// TIA Portal V21 export
TYPE "Std_stMotore"
   STRUCT
      In : Struct
         Setup : Bool;
         CmdPosRich : Bool;
         CmdNegRich : Bool;
         Positioning : Bool;
         PosRelativo : Bool;
         CambioVelDaPunto : Bool;
         ConsMovimentoPos : Bool;
         ConsMovimentoNeg : Bool;
         Premagnetizza : Bool;
         PremagnetizzaPos : Bool;
         PremagnetizzaNeg : Bool;
         ForzaEndLessPos : Bool;
         ForzaEndLessNeg : Bool;
         ForzaEndLessBreve : Bool;
         AttivaLimVarPos : Bool;
         AttivaLimVarNeg : Bool;
         MotoreRun : Bool;
         FrenoSganciato : Bool;
         AnticadutaON : Bool;
         AnticadutaOFF : Bool;
         CinghiaRotta : Bool;
         CoppiaSuperata : Bool;   // Ingresso digitale di coppia superata
         SezAperto : Bool;   // Ingresso digitale per sezionatore motore
         TerMotoreOff : Bool;   // Scatto termico motore
         TerVentolaOff : Bool;   // Scatto termico della servoventola
         DriverFault : Bool;   // Ingresso digitale per fault inverter
         DriverWarning : Bool;
         NoComunInv : Bool;
         NoComunEnc : Bool;
         SensAzz : Bool;
         SpinaSicNoInPos : Bool;
         IngInv01 : Bool;
         IngInv02 : Bool;
         IngInv03 : Bool;
         IngInv04 : Bool;
         IngInv05 : Bool;
         IngInv06 : Bool;
         IngInv07 : Bool;
         IngInv08 : Bool;
         PercentualeRichiesta : Int := 100;
         TrgPos : DInt;
         TrgPosRel : DInt;
         CmdVelocitaRich : DInt;
         Acc : DInt;
         Dec : DInt;
         PosCambioVel : DInt;
         VelCambioVel : DInt;
         LimiteVarPos : DInt;
         LimiteVarNeg : DInt;
         ValoSetupEnc : DInt;
      END_STRUCT;
      HW : Struct
         TipoCollInverter : Int;
         HWIO_Inverter : HW_IO;
         HWIO_Parametri : HW_IO;
         HWIO_Inverter_Out : HW_IO;
         HWIO_Parametri_Out : HW_IO;
         TipoEncoder : Int;
         HWIO_Encoder : HW_IO;
         HWIO_PrmEncoder : HW_IO;
      END_STRUCT;
      Prm : Struct
         Quote : Array[0.."K_NumCamma"] of Real;
         UnitàMisura : "Std_UnitàDiMisura";
         Mech : Struct
            Direction : Bool;
            EndLess : Bool;
            GearIn : UInt;
            GearOut : UInt;
            FeedConstant : UDInt;
            RPMMaxRef : UInt;
            JLoad : DInt;
            Z176 : DInt;
         END_STRUCT;
         Enc : Struct
            Direction : Bool;
            EncoderLess : Bool;
            Z180_2 : Bool;
            Z180_3 : Bool;
            Z180_4 : Bool;
            Z180_5 : Bool;
            Z180_6 : Bool;
            Z180_7 : Bool;
            ModoCalcoloK : Bool;
            SetupDoppio : Bool;
            Z181_2 : Bool;
            Z181_3 : Bool;
            Z181_4 : Bool;
            Z181_5 : Bool;
            Z181_6 : Bool;
            Z181_7 : Bool;
            Mounting : USInt;
            SetupMode : USInt;
            ModuloPosEnc : DInt := DINT#1_000_000_000;
            ModuloNegEnc : DInt;
            KSetup : DInt;
            FeedConstant : UDInt;
            ImpRev : Real;
         END_STRUCT;
         C : Struct
            ContPrema : Int;
            OldPosEncoder : DInt;
            TrgPos : Real;
            SpazioGiroEncoder : Real;
            EncPos : Real;
            VelMax : DInt;
         END_STRUCT;
         "M" : Struct
            RichManPos : Bool;
            RichManNeg : Bool;
            AsseNuovaPosManRich : Bool;
         END_STRUCT;
         AbiltManutenzionePrev : Bool;
         K_Analogica : Int;
         EscludiFunzPos : Bool;
         CalcTempoRimanente : Bool;
         CambioDirNoFreno : Bool;
         PremaNoFreno : Bool;
         FrenoPresente : Bool;
         FBKFrenoPresente : Bool;
         AnticadutaPresente : Bool;
         ByPassAnticaduta : Bool;
         DisabCicloAutoAllarme : Bool;
         DisabCicloManuAllarme : Bool;
         TReazioneSistema : Int := 120;
         TPrema : Int := 250;
         TBassaVel : Int := 100;
         TAggancioFreno : Int := 100;
         TSgancioFreno : Int := 100;
         TOutPrema : Int := 1000;
         TMinVCost : Int;
         TCambioDir : Int;
         ValMaxRef : Int;
         LimitePos : DInt;
         LimiteNeg : DInt;
         PosManutenzione : DInt;
         VelPrema : DInt;
         VelBassa : DInt;
         VelSgancioFrenoPos : DInt;
         VelSgancioFrenoNeg : DInt;
         SpazioArrestoPos : DInt;
         SpazioArrestoNeg : DInt;
         Precisione : DInt;
         Inerzia : DInt;
         FollowingLimit : DInt;
         MaxCopia : DInt;
         DecFinale : DInt;
         DecEmergenza : DInt;
         Jerk : DInt;
         VelMan : DInt;
         VelJog : DInt;
      END_STRUCT;
      Dati : Struct
         BloccoRichiamato : Bool;
         InclusoInUnaSequenza : Bool;
         SetupPN : Struct
            Input : Struct
               REQ : Bool;
               ID : Bool;
               INDEX : Bool;
               LEN : Bool;
            END_STRUCT;
            Output : Struct
               DONE : Bool;
               BUSY : Bool;
               ERROR : Bool;
               STATUS : DWord;
            END_STRUCT;
         END_STRUCT;
         MP : Struct
            SpazioPercorso : DInt;
            TempoMovimento : DInt;
            ImpMarcia : Bool;
            ImpFreno : Bool;
            MetriPercorsi : DInt;
            MinutiLavorati : DInt;
            NAvviamenti : DInt;
            NSgancioFreno : DInt;
         END_STRUCT;
         MotorStop : Bool;
         ActVelPos : Bool;   // Velocità Positiva in Corso
         ActVelNeg : Bool;   // Velocità Negativa in Corso
         MotoreFermo : Bool;   // Motore fermo
         RitAggancioFreno : Bool;   // Memoria tempo aggancio freno trascorso
         CambioDirezioneAlVolo : Bool;   // Eseguito cambio direzione al volo
         SetupSensoreTrovato : Bool;   // Sensore di Setup Trovato
         SetupFermoMeccTrovato : Bool;   // Arresto meccanico durante procedura di Set Up Trovato
         TOffInverterStatus : Bool;   // Ritardo OFF segnale stato inverter
         TOffMotoreMarcia : Bool;   // Ritardo OFF Motore in Marcia
         AppoImpMotoreFermo : Bool;   // Appoggio Impulso motore fermo
         AppoImpEsecSetUP : Bool;   // Appoggio Impulso richiesta SetUP Sensore o Fermo Meccanico
         AppoImpOnSegnSonora : Bool;   // Appoggio Impulso ON Segnalazione Sonora
         AppoImpFunzPositioning : Bool;   // Appoggio Impulso Richiesta funzionamento in posizione
         AppoImpMovRelativo : Bool;   // Appoggio Impulso per richiesta movimento relativo
         AppoImpCaVelPunto : Bool;   // Impulso di cambio velocità da punto
         StatoFreno : Bool;   // Stato Freno
         PrmSend : Bool;
         ContMotoreInPrec : Int;   // Conteggio tempo di motore all'interno della precisione [ms]
         ContTimeOutInverter : Int;   // Contatore Time Out Inverter [ms]
         ContTimeOutFreno1 : Int;   // Contatore Time Out Freno 1 (Rilascio) [ms]
         ContTimeOutFreno2 : Int;   // Contatore Time Out Freno 2 (Sganciato inaspettatamente) [ms]
         ContSgancioFreno : Int;   // Contatore ritardo Sgancio [ms]
         ContAggancioFreno : Int;   // Contatore ritardo Aggancio [ms]
         ContTimeOutPrema : Int;   // Contatore Time Out premagnetizzazione [ms]
         ContTOffInverterStatus : Int;   // Contatore Ritardo OFF Segnale Inverter Status [ms]
         ContTOffMotoreMarcia : Int;   // Contatore Ritardo OFF Motore in Marcia [ms]
         ContCheckFollowError : Int;   // Contatore per il controllo progressivo del Following Error [ms]
         ContSetUPEncoder : Int;   // Contatore per l'esecuzione del SetUP Encoder
         Memo_PercentualeRich : Int;   // Memorizzo la percentuale di velocità richiesta
         ContTimeOutAzzeramento : Int;   // Contatore Time Out Ricerca Sensori Azzeramento [ms]
         ContTOutAnticaduta : Int;   // Contatore Time-Out Anticaduta
         RetVal_Read_Inv : Int;   // Ret Val funzione Lettura Profibus dall'Inverter
         RetVal_SCR_Inv : Int;   // Ret Val funzione Scrittura Profibus all'Inverter
         ContCambioDirPos : Int;   // Contatore per cambio direzione Positiva
         ContCambioDirNeg : Int;   // Contatore per cambio direzione Negativa
         ContOffSezAperto : Int;   // Contatore per controllo sezionatore aperto SEW
         ContSegnSetup : Int;   // Contatore per segnalazione Setup Eseguita
         ContTORichSetup : Int;   // Contatore Time-Out richiesta Setup
         ContAbilAccDopoCambioDir : Int;   // Contatore Abilitazione Accelerazione dopo Cambio Direzione
         ContFermoMeccTrovato : Int;   // Contatore Fermo Meccanico Trovato
         IdPrm : UInt;   // Contatore Scrittura Parametri
         TempoEsecuzioneProfilo : DInt;   // Tempo esecuzione Profilo [ms]
         ContTimeOutMovimento : DInt;   // Contatore Time Out Movimento Motore [ms]
         ChFol_SpazioEncoder : DInt;   // Check Following: Spazio percorso dall'encoder nel tempo di controllo [Unità]
         ChFol_SpazioTarget : DInt;   // Check Following: Spazio percorso dal target nel tempo di controllo [Unità]
         TRG_OLD_POS_Select : DInt;   // OLD Posizione di target filtrata
         PosizioneAlloStop : DInt;   // Memorizzazione della posizione al momento dell'arresto [Unità]
         PosizioneCheckDirezione : DInt;   // Memorizzazione della posizione per il controllo della direzione [Unità]
         VeloRichPerc : DInt;   // Velocità richiesta dopo calcolo percentuale [Unità/s]
         AccRichPerc : DInt;   // Accelerazione richiesta dopo calcolo percentuale [Unità/s/s]
         DecRichPerc : DInt;   // Decelerazione richiesta dopo calcolo percentuale [Unità/s/s]
         VeloDopoCambioRich : DInt;   // Velocità dopo cambio richiesta [Unità/s]
         TrgPosDint : DInt;   // Posizione di target (Valore Intero) [Unità]
         OldTrgPosDint : DInt;   // Ultima Posizione di target (Valore Intero) [Unità]
         OldEncoder : DInt;   // Ultima Posizione letta dell'encoder [Unità]
         Memo_Req_Vel : DInt;   // Memorizzo la velocità richiesta [Unità/s]
         Memo_Req_Acc : DInt;   // Memorizzo l'accelerazione richiesta [Unità/s/s]
         Memo_Req_Dec : DInt;   // Memorizzo la decelerazione richiesta [Unità/s/s]
         Memo_Req_Dec_Emergenza : DInt;   // Memorizzo la decelerazione d'emergenza richiesta [Unità/s/s]
         PosImpulsoSetup : DInt;   // Posizione dell'impulso del sensore di Setup o della posizione di Fermo Meccanico [Unità]
         DecReqInLavo : DInt;   // Decelerazione richiesta in lavorazione
         DecReqFinaleInLavo : DInt;   // Decelerazione finale richiesta in lavorazione
         DecReqEmergInLavo : DInt;   // Decelerazione finale richiesta in lavorazione
         MovRelRichiesto : DInt;   // Movimento relativo richiesto [Unità]
         MemoCheckInversione : DInt;   // Memoria Controllo Inversione
         MaxPosRicercaFermoMeccanico : DInt;   // Massima Posizione durante la ricerca del fermo meccanico
         ReqVelConv : Real;   // Velocità richiesta convertito in REAL [Unità]
         VeloMinConv : Real;   // Velocità minima convertita
         Encoder : Struct
            PrmEncSend : Bool;   // Parametro Encoder Inviati
            OLD_Senso_Rotazione : Bool;   // Appoggio ultimo senso di rotazione Impostato
            RichSetupEnc { ExternalAccessible := 'False'; ExternalVisible := 'False'; ExternalWritable := 'False'} : Bool;   // Richiesta Setup Encoder
            RetValRdEnc : Int;   // RetVal funzione di lettura encoder
            RetValScrEnc : Int;   // RetVal funzione di scrittura encoder
            RicircoloEncoder : DInt := 0;   // Valore di ricircolo Encoder
            MezzoRicircoloEncoder : DInt := 0;   // Valore di mezzo ricircolo Encoder
            o_OldPosEncoder : DInt;   // Ultima posizione Encoder registrata [Impulsi]
            OLD_Spazio_Giro_Encoder : Real;   // Appoggio l'ultimo spazio per giro encoder Impostato
            ValoKSetupSuSens : DInt;   // Valore K Per Setup su Sensore
         END_STRUCT;
         AlmInv_ResetInverter : Bool;   // Allarme Inverter: Reset Inverter
         Alm_ContAzzCont : DInt;   // Autoreset Allarmi: Contatore Azzeramento Contatore Allarmi
         AlmBloccato_Cont : DInt := 0;   // Allarmi Bloccato: Conteggio
         AlmInv_ToutReset : Int;   // Allarme Inverter: Time Out Reset
         AlmInv_Cont : DInt := 0;   // Allarme Inverter: Conteggio
         AlmInv_ContStorico : DInt := 0;   // Allarme Inverter: Conteggio Storico
         AlmInv_RitRestart : Int;   // Allarme Inverter: Ritardo Ripartenza
         AlmInv_StoricoCodici : Array[0..9] of DInt;   // Allarme Inverter: Storico Codici
      END_STRUCT;
      HMI : Struct
         Visibilita : Struct
            Servoventola : Bool;
         END_STRUCT;
         Param : Struct
            Read : Bool;
            Write : Bool;
            Save : Bool;
            FactoryInit : Bool;
            Init_Motor : Bool;
            ReadAll : Bool;
            Number : Int;
            SubNumber : Int;
            Value : DInt;
         END_STRUCT;
         Setup : Bool;
         PulsanteSetupPremuto : Bool;
         ManMov : Bool;
         UpdParam : Bool;
         UM : USInt;
         FBGestione : Int;
         IndexAreaAuto : UInt;
         Stato : USInt;
         ComandoRichiesto : USInt;
         STW1 : Word;
         STW2 : Word;
         STW3 : Word;
         CTW1 : Word;
         CTW2 : Word;
         CTW3 : Word;
         ValoreSetupEncoder : DInt;
         ValoreSetupRichiesto : DInt;
         ValoreSetupSensore : DInt;
         CodiceWarning : DInt;
         CodiceAllarme : DInt;
         ModoInizializza : USInt;
         ALM : Array[0..1] of Word;
      END_STRUCT;
      Allarmi : Struct
         "A" : Array[0.."K_NumAllarmiPerMotori"] of "Std_PrmAllarmeStd";
         WordHmi_1 { S7_SetPoint := 'True'} : Word;
         WordHmi_2 : Word;
         ComunInverter : Bool;
         ComunEncoder : Bool;
         TOutMarcia : Bool;
         ConteggioEnc : Bool;
         FolError : Bool;
         Bloccato : Bool;
         TroppoVeloce : Bool;
         Direzione : Bool;
         EncMismatch : Bool;
         TOUTMovimento : Bool;
         InverterFault : Bool;
         TermicoVentola : Bool;
         RotturaCinghia : Bool;
         TimeOutAnticaduta : Bool;
         Freno : Bool;
         Freno2 : Bool;
         TOUT_Azzeramento : Bool;
         MotoreNonParam : Bool;
         EncoderNonSetup : Bool;
         SetupEncoderEseg : Bool;
         InverterWarning : Bool;
         Parametri : Bool;
         SezAperto : Bool;
         SpinaSicNoInPos : Bool;
         TrgPosMinNeg : Bool;
         TrgPosMaxPos : Bool;
         TrgPosMinNegVar : Bool;
         TrgPosMaxPosVar : Bool;
         AccRichZero : Bool;
         AccRichMaxMaxDec : Bool;
         DecRichZero : Bool;
         DecRichMaxMaxDec : Bool;
         DecFinaleRichZero : Bool;
         DecFinaleRichMaxMaxDec : Bool;
         DecEmergenzaRichZero : Bool;
         TrgVelMinFreno : Bool;
         TrgVelMaxMax : Bool;
         TrgVelCamMinFreno : Bool;
         TrgVelCamMaxMax : Bool;
      END_STRUCT;
      Out : Struct
         Pronto : Bool;
         PremaOK : Bool;
         TOUTPrema : Bool;
         InMarcia : Bool;
         ActDirPos : Bool;
         ActDirNeg : Bool;
         FaseAcc : Bool;
         FaseDec : Bool;
         PosOK : Bool;
         RichMovPos : Bool;
         RichMovNeg : Bool;
         MinLimNeg : Bool;
         MaxLimPos : Bool;
         ActInInerzia : Bool;
         MinTrg : Bool;
         MaxTrg : Bool;
         CmdPosServoventola : Bool;
         CmdPosMotore : Bool;
         CmdNegMotore : Bool;
         CmdAnticaduta : Bool;
         CmdFreno : Bool;
         RitSgancioFreno : Bool;
         Allarme : Bool;
         DisContattori : Bool;
         Lampada : Bool;
         Sirena : Bool;
         EncoderHomed : Bool;
         SetUpSensEseg : Bool;
         UpdParam : Bool;
         CmdUsc01Inv : Bool;
         CmdUsc02Inv : Bool;
         CmdUsc03Inv : Bool;
         CmdUsc04Inv : Bool;
         Paw : Word;
         ActPos : DInt;
         SpazioStop : DInt;
         ActPosPiuStop : DInt;
         ActPosPiuInerzia : DInt;
         ActPosMenoInerzia : DInt;
         SpazioCicloEnc : DInt;
         DistTRG : DInt;
         TrgPosFiltrata : DInt;
         FollowingError : DInt;
         MotorSpeed : DInt;
         TFineProfilo : DInt;
         Vel : Real;
         VelAss : Real;
         VelEncoder : DInt;
      END_STRUCT;
      Rif_Inc : Struct
         K_Pid : Int;
         K_Zona : Int := 0;
         K_Analogica : Int;   // Utilizzato per il feedback speed
         K_Sequenza : Array[0.."K_NumRifIncrociatiSequenza"] of Int;
      END_STRUCT;
   END_STRUCT;
END_TYPE
